(* CoDeSys 2.3 export: MQTT_UDP_USE.EXP *)

(* POU HTTP/MQTT_UDP_PRG, ST *)
PROGRAM MQTT_UDP_PRG
VAR
	MQ		:	MQTT_UDP;
END_VAR
	(* 	MQ_SEND_REAL( MQ, 'Name', Value );  *)

	MQ_SEND_REAL( MQ, 'PLK0_WarmWaterConsumption', GLOBAL_WarmWaterConsumption );
	MQ_SEND_REAL( MQ, 'PLK0_ColdWaterConsumption', GLOBAL_ColdWaterConsumption );

	MQ_SEND_REAL( MQ, 'PLK0_activePa', GLOBAL_activePa_avg * 10 ); 
	MQ_SEND_REAL(  MQ, 'PLK0_Va', Va );
END_PROGRAM
